TYPE ParIDAccess_Input_typ :
	STRUCT
		Command 	: ParIDAccess_CMD_typ ;
		Parameter	: ParIDAccess_Param_typ ;
	END_STRUCT
END_TYPE

(* stored: Version 1.1.0.1, ProductVersion 3.1.4024.3
   DUT ParIDAccess_Input_typ: Id {3f2e5115-52c2-08fc-2905-656b9f029781} *)
